// TIA Portal project "Nadrz" (V15)

(* hardware
DEVICE "S71500/ET200MP station_1"  S7-1500 station
   slot 0: "Rail_0"  Rack  6ES7 590-1***0-0AA0
   slot 1: "s7-1500"  CPU 1515-2 PN  6ES7 515-2AM01-0AB0  V2.5
      slot 3: "CPU display_1"  6ES7591-1BA00-0AA0
   slot 2: "AI 8xU/I HS_1"  AI 8xU/I HS  6ES7 531-7NF10-0AB0  V2.1
   slot 3: "AQ 2xU/I ST_1"  AQ 2xU/I ST  6ES7 532-5NB00-0AB0  V1.0
   slot 4: "DI 16x24VDC BA_1"  DI 16x24VDC BA  6ES7 521-1BH10-0AA0  V1.0
*)

// ===== PLC "s7-1500"  CPU 1515-2 PN =====

VAR_GLOBAL   // PLC tag table "Default tag table"
   "vq1Out" AT %QW0 : Int;
   "vq2Out" AT %QW2 : Int;
   "vq1Fbk" AT %IW10 : Int;
   "vq2Fbk" AT %IW12 : Int;
   "hladina" AT %IW14 : Int;
   "vq2SP" AT %IW16 : Int;
   "hladinaSP" AT %IW18 : Int;
END_VAR

DATA_BLOCK "Data"   // DB2
{ S7_Optimized_Access := 'TRUE' }
VERSION : 0.1
   VAR
      q2_sp : Real;
      q2_real : Real;
      q1_real : Real;
   END_VAR
BEGIN
END_DATA_BLOCK

DATA_BLOCK "Ventily_DB"   // DB3
{ S7_Optimized_Access := 'TRUE' }
VERSION : 0.1
// stored: InstanceOfName Ventily
"Ventily"
BEGIN
END_DATA_BLOCK

ORGANIZATION_BLOCK "Main"   // OB1, LAD, ProgramCycle
TITLE = "Main Program Sweep (Cycle)"
{ S7_Optimized_Access := 'TRUE' }
VERSION : 0.1
   VAR_INPUT
      Initial_Call : Bool;   // Initial call of this OB
      Remanence : Bool;   // =True, if remanent data are available
   END_VAR
BEGIN

REGION Network 1
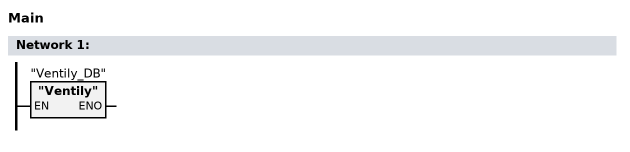
   RUNG wire#powerrail
      "Ventily_DB"()
   END_RUNG
   // the same network as SCL:
   "Ventily_DB"();   // "Ventily"
END_REGION
END_ORGANIZATION_BLOCK

// folder: pristroje/Ventily

FUNCTION_BLOCK "Ventily"   // FB1, LAD
{ S7_Optimized_Access := 'TRUE' }
VERSION : 0.1
   VAR_TEMP
      norm_vq2sp : Real;
   END_VAR
BEGIN

REGION Network 1: vq1
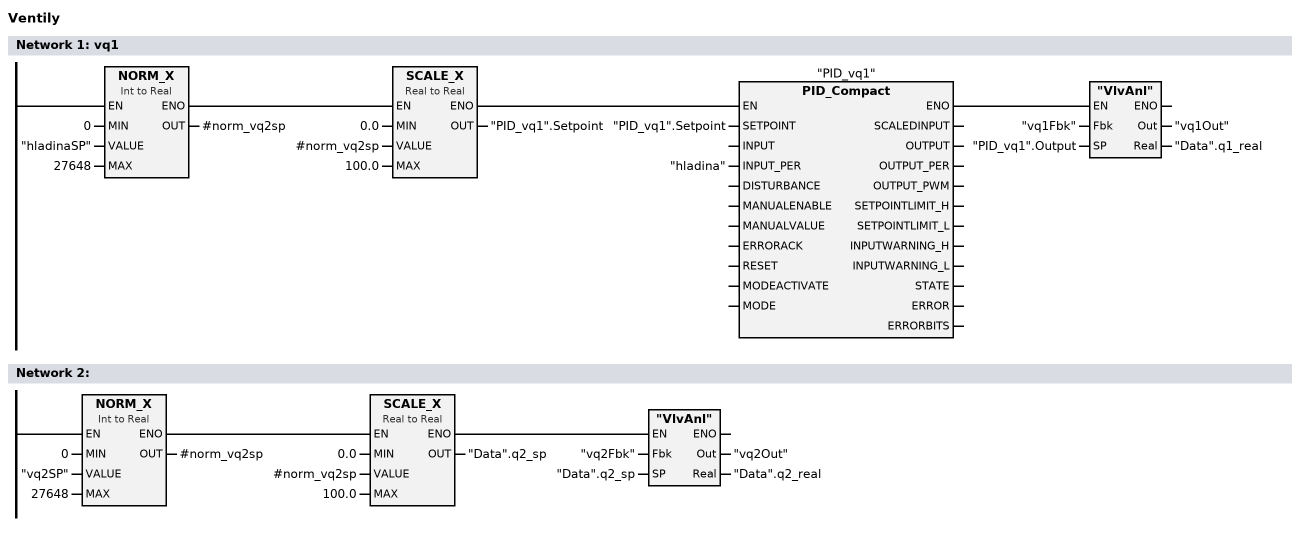
   // ENO of a box is taken as its EN; it also drops when the box reports an error
   #norm_vq2sp := NORM_X(MIN := 0, VALUE := "hladinaSP", MAX := 27648);
   "PID_vq1".Setpoint := SCALE_X(MIN := 0.0, VALUE := #norm_vq2sp, MAX := 100.0);
   "PID_vq1"(Setpoint := "PID_vq1".Setpoint, Input_PER := "hladina");   // PID_Compact
   "VlvAnl"(Fbk := "vq1Fbk", SP := "PID_vq1".Output, Out => "vq1Out", "Real" => "Data".q1_real);
END_REGION

REGION Network 2
   RUNG wire#powerrail
      { S7_Templates := "[SrcType := Int, DestType := Real]" } Normalize(min := 0, value := "vq2SP", max := 27648, out => #norm_vq2sp)
      { S7_Templates := "[SrcType := Real, DestType := Real]" } Scale(min := 0.0, value := #norm_vq2sp, max := 100.0, out => "Data".q2_sp)
      "VlvAnl"(Fbk := "vq2Fbk", SP := "Data".q2_sp, Out => "vq2Out", "Real" => "Data".q2_real)
   END_RUNG
   // the same network as SCL:
   #norm_vq2sp := NORM_X(MIN := 0, VALUE := "vq2SP", MAX := 27648);
   "Data".q2_sp := SCALE_X(MIN := 0.0, VALUE := #norm_vq2sp, MAX := 100.0);
   "VlvAnl"(Fbk := "vq2Fbk", SP := "Data".q2_sp, Out => "vq2Out", "Real" => "Data".q2_real);
END_REGION
END_FUNCTION_BLOCK

FUNCTION "VlvAnl" : Void   // FC1, LAD
{ S7_Optimized_Access := 'FALSE' }
VERSION : 0.1
   VAR_INPUT
      Fbk : Word;
      SP : Real;
   END_VAR
   VAR_OUTPUT
      Out : Word;
      "Real" : Real;
   END_VAR
   VAR_TEMP
      norm_fbk : Real;
      norm_out : Real;
   END_VAR
BEGIN

REGION Network 2: Fbk
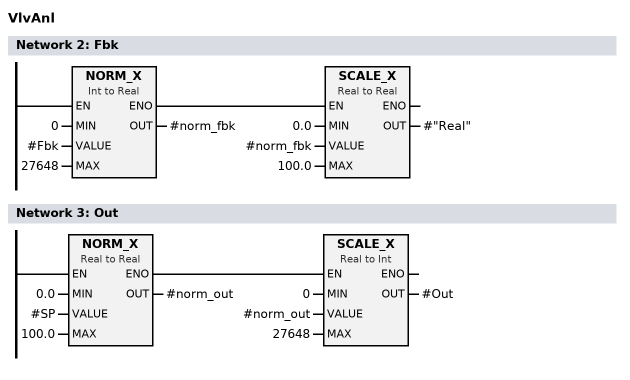
   RUNG wire#powerrail
      { S7_Templates := "[SrcType := Int, DestType := Real]" } Normalize(min := 0, value := #Fbk, max := 27648, out => #norm_fbk)
      { S7_Templates := "[SrcType := Real, DestType := Real]" } Scale(min := 0.0, value := #norm_fbk, max := 100.0, out => #"Real")
   END_RUNG
   // the same network as SCL:
   #norm_fbk := NORM_X(MIN := 0, VALUE := #Fbk, MAX := 27648);
   #"Real" := SCALE_X(MIN := 0.0, VALUE := #norm_fbk, MAX := 100.0);
END_REGION

REGION Network 3: Out
   RUNG wire#powerrail
      { S7_Templates := "[SrcType := Real, DestType := Real]" } Normalize(min := 0.0, value := #SP, max := 100.0, out => #norm_out)
      { S7_Templates := "[SrcType := Real, DestType := Int]" } Scale(min := 0, value := #norm_out, max := 27648, out => #Out)
   END_RUNG
   // the same network as SCL:
   #norm_out := NORM_X(MIN := 0.0, VALUE := #SP, MAX := 100.0);
   #Out := SCALE_X(MIN := 0, VALUE := #norm_out, MAX := 27648);
END_REGION
END_FUNCTION